{attribute addProperty BoxType "KL2541"}
{attribute addProperty Id "Channel_1Channel_866A5B1700"}
{attribute addProperty CRC "4056244207"}
{attribute addProperty SizeInBites "0"}
{attribute addProperty SizeInBytes "0"}
TYPE KL2541_F1C55FEF :
STRUCT
	{attribute addProperty Name "Channel_1"}
	Channel_1 : Channel_866A5B17;
END_STRUCT
END_TYPE

(* stored: Version 1.2.0.0, ProductVersion 3.1.4024.9
   DUT KL2541_F1C55FEF: Id {00214f34-7d64-4f08-90bd-0f60ea553a53} *)
